DATA_BLOCK "bioVal.DB"
{ S7_Optimized_Access := 'TRUE' }
VERSION : 1.0
// Batch I/O Value Data Block:
// by Woermann Automation
NON_RETAIN
   VAR RETAIN
      Val : Array[0..15] of "bioVal.DT";
   END_VAR

BEGIN

END_DATA_BLOCK

